ABB RAPID module: Part_5.mod

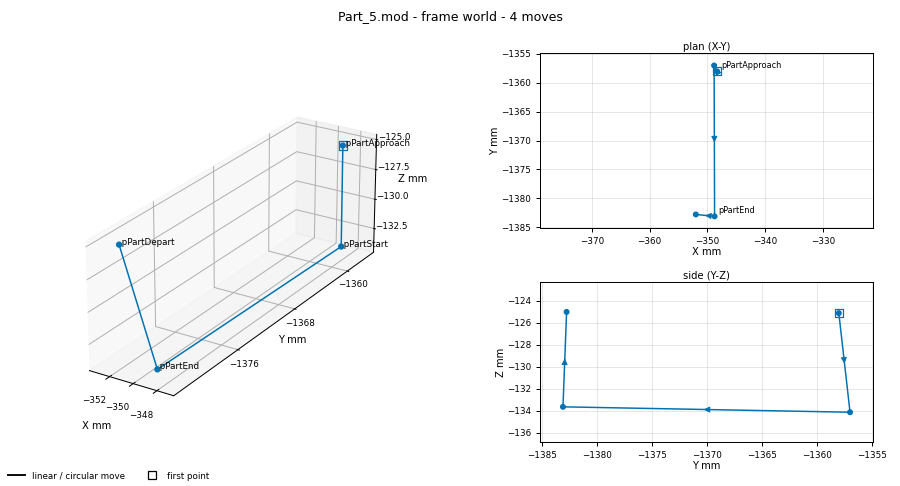
[picture p0: tool path of Part_5.mod in frame world, 4 of 9 moves have a stored position in this frame; points joined in program order, loops and branches not executed]
MODULE Part_5
  ! ------------------------------------------------------------------
  ! Single-part welding template
  !
  ! Purpose:
  !   - Run one part only (no multi-part branching)
  !   - Keep nozzle cleaning and BullsEye tool check available
  !   - Provide a copy/paste starting point for new part files
  !
  ! Dependencies:
  !   - LogicZ (home/safe/pounce positions + rTC2013)
  !   - BE_User1 (BECheckToolb for BullsEye)
  !   - mTSC (optional torch cleaner if you prefer MechCleanGun)
  ! ------------------------------------------------------------------

  PERS bool bUseTorchClean := TRUE;
  PERS bool bUseBullseye := TRUE;

  ! Placeholder weld/seam data for the template. Replace with real values.
  TASK PERS welddata weldPart := [0,0,[1,0,0,0,0,0,0,0,0],[0,0,0,0,0,0,0,0,0]];
  TASK PERS seamdata seamPart := [1,1,[1,0,0,0,0,0,0,0,0],0,0,0,0,0,[0,0,0,0,0,0,0,0,0],0,0,[0,0,0,0,0,0,0,0,0],0,0,[0,0,0,0,0,0,0,0,0],0];

  ! Placeholder targets for the weld path. Replace with taught points.
  CONST robtarget pPartApproach := [[-348.32,-1358.04,-125.11],[0.0288552,0.954843,-0.0190534,0.295092],[-2,-1,1,0],[9E+09,9E+09,9E+09,9E+09,9E+09,9E+09]];
  CONST robtarget pPartStart := [[-348.85,-1357.02,-134.12],[0.0288204,0.95485,-0.0190118,0.295075],[-2,-1,1,0],[9E+09,9E+09,9E+09,9E+09,9E+09,9E+09]];
  CONST robtarget pPartEnd := [[-348.77,-1383.12,-133.63],[0.144948,0.917185,-0.235244,0.287092],[-2,-1,1,0],[9E+09,9E+09,9E+09,9E+09,9E+09,9E+09]];
  CONST robtarget pPartDepart := [[-352.02,-1382.79,-125.00],[0.145009,0.917103,-0.235465,0.287142],[-2,-1,1,0],[9E+09,9E+09,9E+09,9E+09,9E+09,9E+09]];
  PROC RunPart_5()
    TPWrite "Single-part template start";

    ! Optional BullsEye tool check before running a part.
    IF bUseBullseye THEN
      BECheckToolb;
    ENDIF

    ! Optional nozzle cleaning/reaming before the part weld.
    IF bUseTorchClean THEN
      rTC2013;
      ! Alternative: MechCleanGun;  ! From mTSC.mod
    ENDIF

    MoveJ LogicZ::pHomePos, v800, fine, tWeldGun;
    MoveJ LogicZ::pSafeS1, v800, fine, tWeldGun;
    MoveJ LogicZ::pPounceS1, v800, fine, tWeldGun;

    ! ----------------------------------------------------------------
    ! Single-part weld path (edit only the weld start/end points).
    ! ----------------------------------------------------------------
    MoveL pPartApproach, v200, z10, tWeldGun;
    ArcLStart pPartStart, v30, seamPart, weldPart, fine, tWeldGun;
    ArcLEnd pPartEnd, v30, seamPart, weldPart, fine, tWeldGun;
    MoveL pPartDepart, v200, z10, tWeldGun;

    MoveJ LogicZ::pSafeS1, v800, fine, tWeldGun;
    MoveJ LogicZ::pHomePos, v800, fine, tWeldGun;

    TPWrite "Single-part template complete";
  ENDPROC
ENDMODULE
